Universal Robots PolyScope program: urpclientprogram.urp

Program URClient (createdIn=3.4.5.437 lastSavedIn=3.4.5.437 directory=/programs/URClient installation=default robotSerialNumber=2017307081)
Calibrated DH parameters: a=[0.000065, -0.609605, -0.569684, 0.000059, 0.000099, 0]; d=[0.128194, 4.336054, 1.236291, -5.409118, 0.11576, 0.092314]; alpha=[1.570898, -0.013944, -0.007792, 1.5711, -1.5712, 0]; deltaTheta=[0.006367, -0.089589, 0.029531, 0.074964, 0.034815, -0.025455]
BeforeStart
  socket := socket_open("192.168.15.21", 1025)
  Loop While (checkContinuously=false) expression=socket≟ False
    socket := socket_open("192.168.15.21", 1025)
  position := get_actual_joint_positions()
  Script: socket_send_string(position)
  Script: socket_close()
Robot Program (runOnlyOnce=false motionType=MoveJ speed=1.047198 acceleration=1.396263 useActiveTCP=false)
  Wait Sleep waitTime=0.5
